// TIA Portal V15.1 export
// export: Created 2020-06-12T07:35:53.3037109Z, ExportSetting None, DisplayName Totally Integrated Automation Portal, DisplayVersion V15.1, DisplayName TIA Portal Openness, DisplayVersion V15.1, DisplayName STEP 7 Professional, DisplayVersion V15.1, DisplayName STEP 7 Safety, DisplayVersion V15.1, DisplayName WinCC Advanced, DisplayVersion V15.1
FUNCTION "MELT_ElcMgr" : Void   // FC124, FBD
{ S7_Optimized_Access := 'TRUE' }
// stored: SetENOAutomatically False
   VAR_TEMP
      _reset_tara : Bool;
      _limit : Bool;
      _Wt_pres : Real;
      _hood_area : Real;
      _netto : Real;
      tReqTaraSet : Bool;
      tReqTaraReset : Bool;
   END_VAR
BEGIN

REGION Network 1: HMI request treat
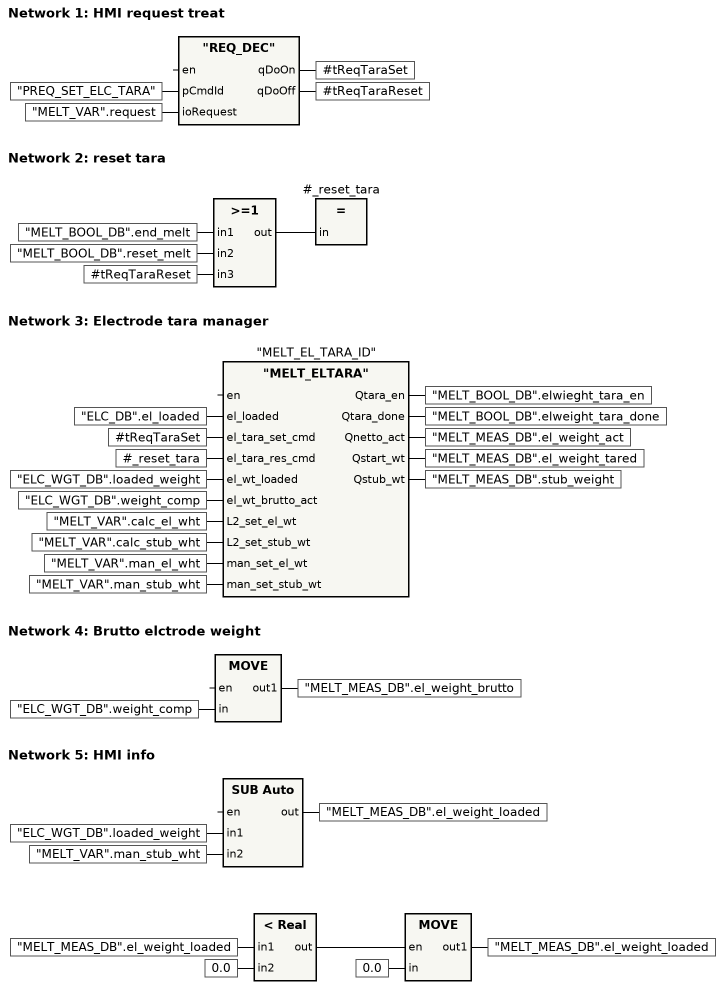
   "REQ_DEC"(pCmdId := "PREQ_SET_ELC_TARA",
             ioRequest := "MELT_VAR".request,
             qDoOn => #tReqTaraSet,
             qDoOff => #tReqTaraReset);
END_REGION

REGION Network 2: reset tara
   #_reset_tara := "MELT_BOOL_DB".end_melt OR "MELT_BOOL_DB".reset_melt OR #tReqTaraReset;
END_REGION

REGION Network 3: Electrode tara manager
   // "MELT_BOOL_DB".elweight_tara_done
   "MELT_EL_TARA_ID"(el_loaded := "ELC_DB".el_loaded,   // "MELT_ELTARA"
                     el_tara_set_cmd := #tReqTaraSet,
                     el_tara_res_cmd := #_reset_tara,
                     el_wt_loaded := "ELC_WGT_DB".loaded_weight,
                     el_wt_brutto_act := "ELC_WGT_DB".weight_comp,
                     L2_set_el_wt := "MELT_VAR".calc_el_wht,
                     L2_set_stub_wt := "MELT_VAR".calc_stub_wht,
                     man_set_el_wt := "MELT_VAR".man_el_wht,
                     man_set_stub_wt := "MELT_VAR".man_stub_wht,
                     Qtara_en => "MELT_BOOL_DB".elwieght_tara_en,
                     Qtara_done => "MELT_BOOL_DB".elweight_tara_done,
                     Qnetto_act => "MELT_MEAS_DB".el_weight_act,
                     Qstart_wt => "MELT_MEAS_DB".el_weight_tared,
                     Qstub_wt => "MELT_MEAS_DB".stub_weight);
END_REGION

REGION Network 4: Brutto elctrode weight
   "MELT_MEAS_DB".el_weight_brutto := "ELC_WGT_DB".weight_comp;
END_REGION

REGION Network 5: HMI info
   "MELT_MEAS_DB".el_weight_loaded := "ELC_WGT_DB".loaded_weight - "MELT_VAR".man_stub_wht;
   IF "MELT_MEAS_DB".el_weight_loaded < 0.0 THEN "MELT_MEAS_DB".el_weight_loaded := 0.0; END_IF;
END_REGION
END_FUNCTION
